Staubli VAL3: decompose_wait.pgx

public program decompose_wait(string& x_sItem[] (dimensions=1), string& x_sName (dimensions=1), num& x_nOperator (dimensions=1), num& x_nValue (dimensions=1))
  local num i
  local num l_nPos
  local num l_nSize
  local string l_sItem
  local bool l_bOk
  local string l_sItem2
begin
  //
  // decompose into Index-Operator-Value-Mode
  //
  for i=0 to size(sCondition)-1
    // Operator
    l_nPos=find(x_sItem,sCondition[i])
    if l_nPos!=-1
      x_nOperator=i
      i=size(sCondition)-1
    endIf
  endFor
  if l_nPos!=-1
    // find the Index
    call getSize_num(l_nSize)
    for i=0 to l_nSize-1
      // search it
      call get_num(l_sItem,i)
      if l_sItem==left(x_sItem,l_nPos)
        x_sName=l_sItem
        i=l_nSize-1
      endIf
    endFor
    // get the value
    toNum(right(x_sItem,len(x_sItem)-l_nPos-2),x_nValue,l_bOk)
    if !l_bOk
      // found the value
      l_sItem2=right(x_sItem,len(x_sItem)-l_nPos-len(sCondition[1]))
      if size(x_sItem)>1
        x_sItem[1]=l_sItem
      endIf
      for i=0 to l_nSize-1
        // search it
        call get_num(l_sItem,i)
        if l_sItem==l_sItem2
          call getValue_num(x_nValue,l_sItem)
          return
        endIf
      endFor
    endIf
  else
    x_sName=""
  endIf
end
